RoboDK station: UR5Trajectory2.rdk

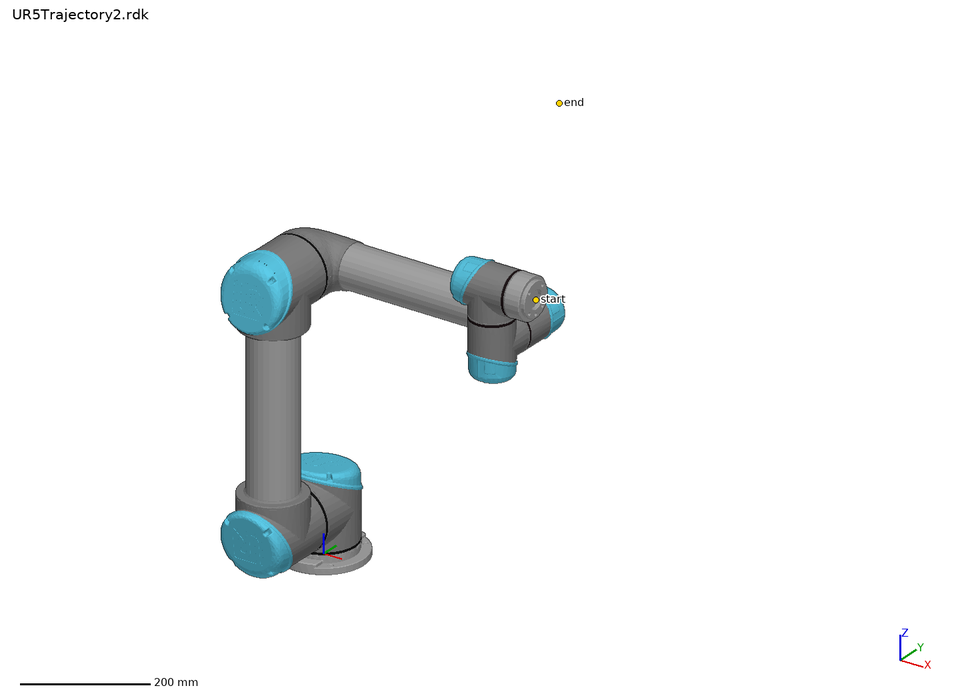
[picture v0: the station drawn from its stored meshes, robots at their saved joint values, targets as dots, program paths as lines]
Station 4TrajectoryUR5 (saved by RoboDK 5.7.0). Poses are relative to the parent item; angles as X-Y-Z fixed-axis rotations.
Station parameters (name, value as stored): test, 7, IO_5, 1, 2, 1, IO_2, 1, digital_out0, 1
  - frame UR5 Base at (0, 0, 0) mm
    - robot UR5: 6 axes
        modified DH rows (alpha deg, a mm, theta deg, d mm): 0, 0, 0, 89.2; 90, 0, 180, 0; 0, 425, 0, 0; 0, 392, 0, 109.3; -90, 0, 0, 94.75; 90, 0, 180, 82.5
        joint limits [-360, -360, -360, -360, -360, -360] to [360, 360, 360, 360, 360, 360]; home [0, -90, -90, 0, 90, 0]; saved at [0, -90, -90, 0, 90, 0]
    - target start (Cartesian target) at (474.5, -109.3, 608.95) mm, rotated rx -90 ry 0 rz -90 deg; joints [0, -90, -90, 0, 90, 0] of UR5
    - target end (Cartesian target) at (109.3, 474.5, 608.95) mm; joints [90, -115.176, -57.109, 82.285, 90, 0] of UR5
    - target Target1 (Cartesian target) at (109.3, 474.5, 608.95) mm; joints [90, -173.574, 89.809, 173.764, -90, -180] of UR5
    - target Target2 (Cartesian target) at (109.3, 474.5, 608.95) mm; joints [90, -169.767, 57.109, 22.658, 90, 0] of UR5
    - target Target3 (Cartesian target) at (109.3, 474.5, 608.95) mm; joints [90, -115.176, -57.109, 82.285, 90, 0] of UR5
    - target Target4 (Cartesian target) at (109.3, 474.5, 608.95) mm; joints [90, -88.375, -89.809, -91.816, -90, -180] of UR5
    - target Target5 (Cartesian target) at (109.3, 474.5, 608.95) mm; joints [244.057, -91.625, 89.809, -88.184, 90, -154.057] of UR5
    - target Target6 (Cartesian target) at (109.3, 474.5, 608.95) mm; joints [244.057, -64.824, 57.109, 97.715, -90, 25.943] of UR5
    - target Target7 (Cartesian target) at (109.3, 474.5, 608.95) mm; joints [244.057, -10.233, -57.109, 157.342, -90, 25.943] of UR5
    - target Target8 (Cartesian target) at (109.3, 474.5, 608.95) mm; joints [244.057, -6.426, -89.809, 6.236, 90, -154.057] of UR5
  - program Start->end1 (1 instructions, listed below)
  - program Start->end2 (1 instructions, listed below)
  - program Start->end3 (1 instructions, listed below)
  - program Start->end4 (1 instructions, listed below)
  - program Start->end5 (1 instructions, listed below)
  - program Start->end6 (1 instructions, listed below)
  - program Start->end7 (1 instructions, listed below)
  - program Start->end8 (1 instructions, listed below)
  - program moveL_Start->end (1 instructions, listed below)
  - program Prog10 (2 instructions, listed below)
  - program Prog11 (1 instructions, listed below)

--- program Start->end1 (robot UR5) ---
  MoveJ (Target1)

--- program Start->end2 (robot UR5) ---
  MoveJ (Target2)

--- program Start->end3 (robot UR5) ---
  MoveJ (Target3)

--- program Start->end4 (robot UR5) ---
  MoveJ (Target4)

--- program Start->end5 (robot UR5) ---
  MoveJ (Target5)

--- program Start->end6 (robot UR5) ---
  MoveJ (Target6)

--- program Start->end7 (robot UR5) ---
  MoveJ (Target7)

--- program Start->end8 (robot UR5) ---
  MoveJ (Target8)

--- program moveL_Start->end (robot UR5) ---
  MoveL (Target8)

--- program Prog10 (robot UR5) ---
  MoveJ (start)
  Set speed (10.0 mm/s)

--- program Prog11 (robot UR5) ---
  Set speed (10.0 mm/s)
